{attribute 'GeneratedUsingTerminal: EPP2316-0003-0016'}
{attribute addProperty BoxType "EPP2316-0003-0016"}
{attribute addProperty Id "Set_safe_stateAT %Q*BOOL1Reset_outputsAT %Q*BOOL1"}
{attribute addProperty CRC "916844311"}
{attribute addProperty Size "2"}
TYPE DIG_Outputs_Device_36A5EF17 :
STRUCT
	{attribute addProperty Name "Set_safe_state"}
	Set_safe_state AT %Q* : BOOL;
	{attribute addProperty Name "Reset_outputs"}
	Reset_outputs AT %Q* : BOOL;
END_STRUCT
END_TYPE

(* stored: Version 1.2.0.0, ProductVersion 3.1.4024.9
   DUT DIG_Outputs_Device_36A5EF17: Id {22ad2ff1-1ee5-43c9-abd5-2b1cf72fa8f8} *)
